Staubli VAL3: pushMotion.pgx

public program pushMotion(num& x_nMsgRecvState)
  local bool l_bOk
  local bool l_bWillMove
  local num l_nCounter
  local num l_nJointError
  local MotionCmd l_mTrajPt
begin
  // Copyright (c) 2016, Ocado Technology - Robotics Research Team
  //
  // Licensed under the Apache License, Version 2.0 (the "License");
  // you may not use this file except in compliance with the License.
  // You may obtain a copy of the License at
  //
  //     http://www.apache.org/licenses/LICENSE-2.0
  //
  // Unless required by applicable law or agreed to in writing, software
  // distributed under the License is distributed on an "AS IS" BASIS,
  // WITHOUT WARRANTIES OR CONDITIONS OF ANY KIND, either express or implied.
  // See the License for the specific language governing permissions and
  // limitations under the License.

  // MoveType = 10: movej(jointRx)
  // MoveType = 20: movej(pointRx)
  // MoveType = 21: movel(pointRx)

  switch rosGenericMsg.header.nMsgType
    case 11
      l_mTrajPt.nMoveType = 10
      l_mTrajPt.nSequence=rosTrajPtMsg.jointTrajPt.nSeq

      // ROS joint position values are in rad, but VAL3 uses degrees
      call toJointRxDeg(rosTrajPtMsg.jointTrajPt.nJoints, l_mTrajPt.jJointRx)

      // from industrial_robot_client/src/joint_trajectory_interface.cpp
      // JointTrajectoryInterface::trajectory_to_msgs()
      // JointTrajectoryInterface::calc_speed()
      // velocity is converted to a scalar value representing % of max velocity,
      // such that 0.2 = 20% of maximum joint speed
      l_mTrajPt.mDesc.vel= limit((rosTrajPtMsg.jointTrajPt.nVelocity * 100), 0, 100)
      l_mTrajPt.nDuration=rosTrajPtMsg.jointTrajPt.nDuration

    break
    case 14
      l_mTrajPt.nMoveType = 10
      l_mTrajPt.nSequence=rosTrajPtFMsg.jointTrajPtFull.nSeq
      l_mTrajPt.nDuration=rosTrajPtFMsg.jointTrajPtFull.nTime

      // ROS joint position values are in rad, but VAL3 uses degrees
      call toJointRxDeg(rosTrajPtFMsg.jointTrajPtFull.nPositions, l_mTrajPt.jJointRx)

      // from industrial_robot_client/src/joint_trajectory_interface.cpp
      // JointTrajectoryInterface::trajectory_to_msgs()
      // JointTrajectoryInterface::calc_speed()
      // velocity is converted to a scalar value representing % of max velocity,
      // such that 0.2 = 20% of maximum joint speed
      l_mTrajPt.mDesc.vel= limit((rosTrajPtFMsg.jointTrajPtFull.nVelocities[0] * 100), 0, 100)
      // not sure about accelerations as yet
      l_mTrajPt.mDesc.accel=rosTrajPtFMsg.jointTrajPtFull.nAccelerations[0]
      l_mTrajPt.mDesc.decel=l_mTrajPt.mDesc.accel
    break
    case 31
      l_mTrajPt.nMoveType = 21
      l_mTrajPt.nSequence=rosTrajPtCartesianMsg.cartesianTrajPt.nSeq

      // ROS position is in meters but VAL3 uses millimeters
      call toPointRxMillis(rosTrajPtCartesianMsg.cartesianTrajPt.nPosition, l_mTrajPt.pPointRx)

      // ROS orientation is in quaternion (rad) but VAL3 uses euler angles
      call toPointRxEuler(rosTrajPtCartesianMsg.cartesianTrajPt.nOrientation, l_mTrajPt.pPointRx)

      // Read accel/decel values
      l_mTrajPt.mDesc.accel = limit(rosTrajPtCartesianMsg.cartesianTrajPt.nAcceleration, 0, 100)
      l_mTrajPt.mDesc.decel = l_mTrajPt.mDesc.accel

      // velocity is a scalar value representing % of max velocity,
      // such that 0.2 = 20% of maximum joint speed
      l_mTrajPt.mDesc.vel= limit((rosTrajPtCartesianMsg.cartesianTrajPt.nVelocity * 100), 0, 100)
      l_mTrajPt.nDuration=rosTrajPtMsg.jointTrajPt.nDuration

    break
    default
    break
  endSwitch

  // see github.com/ros-industrial/industrial_core/simple_message/include/simple_message/joint_traj_pt.h
  if (l_mTrajPt.nSequence==-4)
    // set flag to stop immediately
    bStopNow=true
  else
    // check whether velocity value should be overwritten with value set on teach pendant
    if (bOverwriteVel == true)
      // overwrite velocity (and acceleration - ?)
      l_mTrajPt.mDesc.vel = getMonitorSpeed()
      // explicitly setting accel and decel to VAL3 default values
      l_mTrajPt.mDesc.accel = 9999
      l_mTrajPt.mDesc.decel = 9999
    endIf
    // only push motion into buffer if not a STOP message
    // if it's a joint type of move
    //   and if joint positions are within software joint limits
    //   and if velocity is greater than zero (because movej() will not accept vel <= 0)
    // or if it's a point type of move
    //   and if velocity is greater than zero
    l_bWillMove = false
    if (l_mTrajPt.nMoveType >= 10 and l_mTrajPt.nMoveType < 20) and (isInRange(l_mTrajPt.jJointRx) and l_mTrajPt.mDesc.vel > 0)
      l_bWillMove = true
    elseIf (l_mTrajPt.nMoveType >= 20 and l_mTrajPt.nMoveType < 30) and l_mTrajPt.mDesc.vel > 0
      l_bWillMove = true
    endIf

    if (l_bWillMove == true)

      // Check if we need to power up before the first point of a sequence
      // This is only possible in remote mode.
      if (l_mTrajPt.nSequence == 0)
        // before move, check if we need to enable power
        // (only works if robot is in remote mode)
        if (workingMode() >= 4 and !isPowered())
            do
            enablePower()
            delay(1)
            until isPowered()
        endIf
      endIf

      call libQueueFuncs:push(qTrajPtBuffer,l_mTrajPt,l_bOk)
    else
      l_bOk = false
    endIf

    if (l_bOk==false)
      // could not push trajectory point into buffer
      // thus ACK should flag FAILURE, but only if comm type is request
      if (rosGenericMsg.header.nCommType==2)
        switch rosGenericMsg.header.nMsgType
          case 11
            rosTrajPtAck.header.nReplyCode=2
          break
          case 14
            rosTrajPtFAck.header.nReplyCode=2
          break
          case 31
            rosTrajPtCartesianAck.header.nReplyCode=2
          break
          default
          break
        endSwitch
      endIf
    endIf
  endIf
  // check whether ACK should be sent
  if (rosGenericMsg.header.nCommType == 2)
    // comm type request requires ACK
    x_nMsgRecvState = 5
  else
    // other comm types (e.g., topic) does not require ACK, hence skip state
    x_nMsgRecvState = 0
  endIf
end
